/// This struct contains variables that
/// * are read from outside (e.g. HMI) to retrieve information about the unit's current state and (temporary) parameters (= `publish`) 
/// * are written from outside (e.g. HMI) to control the unit via ADS (= `subscribe`) 
TYPE MachineCom :
STRUCT
  Publish : MachineComPublish;
  Subscribe : MachineComSubscribe;
END_STRUCT
END_TYPE

(* stored: Version 1.1.0.1
   DUT MachineCom: Id {6ba9c5c8-f8ba-4a7e-bfd4-e34f0d317851} *)
